FUNCTION_BLOCK RandomGaussian IMPLEMENTS IRandom
VAR
  _mu : LREAL;
  _sigma : LREAL;    
  _rnd : Tc2_System.DRAND;
END_VAR

METHOD FB_init : BOOL
VAR_INPUT
	bInitRetains : BOOL; // if TRUE, the retain variables are initialized (warm start / cold start)
	bInCopyCode : BOOL;  // if TRUE, the instance afterwards gets moved into the copy code (online change)
  seed : INT;  
  mu : LREAL;
  sigma : LREAL;
END_VAR
SetSeed(seed);
SetMean(mu);
SetSigma(sigma);
END_METHOD

/// Implementation of the Box-Muller transform for normal distributed random
/// variables. There are much faster methods for doing this.
/// Implementation taken from [here](https://en.wikipedia.org/wiki/Box%E2%80%93Muller_transform)
METHOD Next : LREAL
VAR
  u1, u2 : LREAL;
END_VAR
VAR CONSTANT
  Pi : LREAL := 3.14159265358979323846;
END_VAR
//create two random numbers, make sure u1 is greater than epsilon
REPEAT
  _rnd(Num => u1);
  _rnd(Num => u2);  
UNTIL u1 > 1E-8 END_REPEAT

//compute z0 and z1
Next  := (_sigma * SQRT(-2.0 * LOG(u1))) * COS(2*Pi * u2) + _mu;

// we do not need the 2nd randomly distributed variable
// z1 := mag * SIN(2*Struckig.Constants.Pi  * u2) + mu;
END_METHOD

METHOD FINAL SetMean
VAR_INPUT
  mu : LREAL;
END_VAR
_mu := mu;
END_METHOD

METHOD FINAL SetSeed
VAR_INPUT
  seed : INT;
END_VAR
_rnd.Seed := seed;
END_METHOD

METHOD FINAL SetSigma
VAR_INPUT
  sigma : LREAL;
END_VAR
_sigma := sigma;
END_METHOD

END_FUNCTION_BLOCK

(* stored: Version 1.1.0.1
   POU RandomGaussian: Id {f867848b-9e99-4c77-ad60-d50f0ee9a8da}, SpecialFunc None
   Method FB_init: Id {c4f8b591-bc5f-4e63-b859-a1d0657be1db}
   Method Next: Id {a5680f19-16f6-42de-83b9-4823a006e852}
   Method SetMean: Id {774f7473-1d66-48f8-86d9-eb347068eac4}
   Method SetSeed: Id {9b9df88d-eb58-400d-9a6f-dbb295df957c}
   Method SetSigma: Id {1af195a2-705c-43e2-a184-66ec83162e53} *)
